// TIA Portal V20 export
DATA_BLOCK "PM02"   // DB217
// stored: MemoryReserve 100
   VAR
      "C05 UNWINDER SPLICER RIGHT ELECTRODE FIX RIGHT TOP FORWARD" : Bool;
      "C05 UNWINDER SPLICER RIGHT ELECTRODE FIX RIGHT TOP BACKWARD" : Bool;
      "C06 UNWINDER SPLICER RIGHT ELECTRODE FIX RIGHT BTM FORWARD" : Bool;
      "C06 UNWINDER SPLICER RIGHT ELECTRODE FIX RIGHT BTM BACKWARD" : Bool;
      "C07 UNWINDER SPLICER RIGHT CUTTER FORWARD" : Bool;
      "C07 UNWINDER SPLICER RIGHT CUTTER BACKWARD" : Bool;
      "C08 UNWINDER SPLICER LEFT ELECTRODE FIX LEFT TOP FORWARD" : Bool;
      "C08 UNWINDER SPLICER LEFT ELECTRODE FIX LEFT TOP BACKWARD" : Bool;
      "C09 UNWINDER SPLICER LEFT ELECTRODE FIX LEFT BTM FORWARD" : Bool;
      "C09 UNWINDER SPLICER LEFT ELECTRODE FIX LEFT BTM BACKWARD" : Bool;
      "C10 UNWINDER SPLICER LEFT ELECTRODE FIX LEFT TOP DOWN" : Bool;
      "C10 UNWINDER SPLICER LEFT ELECTRODE FIX LEFT TOP UP" : Bool;
      "C11 UNWINDER SPLICER LEFT ELECTRODE FIX LEFT BTM UP" : Bool;
      "C11 UNWINDER SPLICER LEFT ELECTRODE FIX LEFT BTM DOWN" : Bool;
      SPARE_1 : Bool;
      SPARE_2 : Bool;
   END_VAR
BEGIN
END_DATA_BLOCK
